FUNCTION_BLOCK ErrorsWarnings
VAR_INPUT
END_VAR
VAR_OUTPUT
END_VAR
VAR
	CompressorNotRunning: BOOL;
	LineBackedUp: BOOL;
	BeltWrongDirection: BOOL;
	TableWrongDirection: BOOL;
END_VAR

// ERRORS
CompressorNotRunning := NOT gvl.MotorCompressor;
	

//WARNINGS
LineBackedUp := NOT gvl.FotocellOutput;
BeltWrongDirection := gvl.MotorBeltDirection;
TableWrongDirection := gvl.MotorTableDirection;

END_FUNCTION_BLOCK

(* stored: Version 1.1.0.1, ProductVersion 3.1.4024.12
   POU ErrorsWarnings: Id {4bc88007-fc33-4b68-bf49-9f55719a9747}, SpecialFunc None *)
